// SIMATIC S7-200 project (STEP 7-Micro/WIN), CPU 226 CN REL 02.01

ORGANIZATION_BLOCK main:OB1
TITLE=自动化焊接工作站的控制程序。
// 工作站集成了传送带、预热区、焊接区和冷却区。
// 系统由启动按钮触发运行，置位运行状态标志，并通过停止按钮随时中止操作。运行状态标志只有在启动按钮被按下时才能置位，且在停止按钮按下时必须复位，确保操作员对系统状态的完全掌控。
// 焊接过程从工件传送开始。传送带电机将工件送入工作站，但只有在系统运行、工件到位传感器1和工件到位传感器2检测到工件就位，且无错误标志3、错误标志4或错误标志5时才会启动，避免工件缺失或系统故障时的误动作。
// 工件到达预热区后，预热器1开始工作，其激活条件是系统运行、特定信号满足、工件到位传感器1和工件到位传感器2确认工件到位，且无错误标志3或错误标志4，保证预热过程安全进行。预热器2在预热阶段辅助加热。预热器3在另一阶段辅助加热。预热器4在后续阶段辅助加热，以确保工件温度均匀。
// 温度控制是焊接质量的关键。系统通过温度传感器1、温度传感器2和温度传感器3实时监测预热区、焊接区和冷却区的温度，并将读数存储到温度存储变量1~3中。加热器在特定信号为1时启动。加热器应在温度低于设定值且特定信号为真时启动，以维持焊接区适宜温度。加热器在特定信号激活时开始运行。
// 焊接头和喷雾器分别在特定条件下执行操作。喷雾器需在焊接完成后启动，以冷却工件。喷雾器在特定信号触发时启动。
BEGIN
Network 1 // 网络标题
// 网络注释
LD     SM0.0
CALL   preheat1:SBR0
Network 2
LD     SM0.0
CALL   timepulse:SBR1
Network 3
LD     SM0.0
CALL   conveyor:SBR2
Network 4
LD     SM0.0
CALL   xilu:SBR3
Network 5
LD     SM0.0
CALL   preheat4:SBR4
Network 6
LD     SM0.0
CALL   pray:SBR5
Network 7
LD     SM0.0
CALL   preheat2:SBR7
Network 8
LD     SM0.0
CALL   preheat3:SBR8
Network 9
LD     SM0.0
CALL   STARTTIME:SBR9
Network 10
LD     SM0.0
CALL   state:SBR10
Network 11
LD     SM0.0
CALL   wave:SBR11
Network 12
LD     SM0.0
CALL   redlight:SBR6
Network 13
LD     SM0.0
CALL   alarm:SBR12
Network 14
LD     M20.0
EU
S      V0.0, 1
Network 15
LD     M20.1
EU
R      V0.0, 1
Network 16
LD     M20.0
TON    T120, +5
A      T120
R      M20.0, 1
Network 17
LD     M20.1
TON    T121, +5
A      T121
R      M20.1, 1
Network 18
LD     M20.2
EU
O      M0.0
AN     M20.3
AN     V828.0
AN     V828.1
AN     V880.0
=      M0.0
Network 19
LD     M20.2
TON    T122, +5
A      T122
R      M20.2, 1
Network 20
LD     M20.3
TON    T123, +5
A      T123
R      M20.3, 1
Network 21
LDN    V0.0
A      M21.7
O      V0.0
A      M0.0
A      I0.6
A      I0.7
AN     V828.4
AN     V828.2
AN     V830.1
=      Q2.5
Network 22
LD     M22.0
A      M0.0
A      I0.6
A      I0.7
AN     V828.4
AN     V828.2
=      Q1.7
Network 23
LDN    V0.0
A      M22.2
O      V0.0
A      M0.0
A      I0.6
A      I0.7
AN     V828.4
AN     V828.2
AN     V830.6
=      Q2.4
Network 24
LDN    M0.0
R      M20.5, 14
R      M22.4, 1
Network 25
LD     V0.0
R      M20.5, 5
R      M22.1, 2
R      M21.5, 1
R      M22.4, 1
Network 26
LD     V0.0
LD     M20.7
O      M21.0
O      M21.1
O      M21.2
AN     V0.0
OLD
A      M0.0
A      I0.6
A      I0.7
AN     V828.4
AN     V828.2
=      Q2.1
Network 27
LD     M22.5
=      Q0.2
Network 28
LD     M0.0
A      I0.0
EU
+I     +1, VW818
Network 29
LD     M22.3
MOVW   +0, VW818
Network 30
LD     M22.3
TON    T124, +5
A      T124
R      M22.3, 1
Network 31
LD     M22.6
MOVW   AIW10, VW812
MOVW   AIW12, VW814
MOVW   AIW14, VW816
Network 32
LD     M22.7
R      M22.6, 2
R      V822.6, 1
Network 33
LD     M22.6
=      Q1.3
S      V822.6, 1
END_ORGANIZATION_BLOCK

SUBROUTINE_BLOCK preheat1:SBR0
TITLE=子程序注释
BEGIN
Network 1 // 网络标题
// 网络注释
LD     SM0.0
MOVW   VW610, VW1500
MOVW   VW612, VW1502
MOVW   VW614, VW1504
MOVW   VW616, VW1506
Network 2
LD     SM0.0
MOVW   AIW0, VW1508
+I     VW1506, VW1508
Network 3
LDW>=  VW1508, +0
AW<=   VW1508, +2500
MOVW   VW1500, VW1510
+I     +20, VW1510
MOVW   VW1500, VW1512
+I     +5, VW1512
MOVW   VW1500, VW1514
-I     +10, VW1514
MOVW   VW1500, VW1516
-I     +15, VW1516
MOVW   VW1500, VW1518
-I     +20, VW1518
MOVW   VW1500, VW1520
-I     +25, VW1520
MOVW   VW1500, VW1522
-I     +50, VW1522
MOVW   VW1500, VW1524
-I     +100, VW1524
MOVW   VW1500, VW1542
+I     +100, VW1542
Network 4
LD     M12.0
MOVW   VW1508, VW1526
Network 5
LD     M12.2
AW>=   VW1508, VW1526
MOVW   VW1508, VW1528
-I     VW1526, VW1528
Network 6
LDW<=  VW1508, VW1524
LDW<=  VW1508, VW1526
AW<=   VW1508, VW1512
OLD
LD     M15.0
AW<=   VW1508, VW1522
AW>=   VW1508, VW1524
OLD
LD     M15.1
AW<=   VW1508, VW1520
AW>=   VW1508, VW1522
OLD
LD     M15.2
AW<=   VW1508, VW1516
AW>=   VW1508, VW1520
OLD
LDW>   VW1528, +3
A      M15.4
LDW>=  VW1528, +0
AW<=   VW1528, +3
A      M15.5
OLD
AW<=   VW1508, VW1500
AW>=   VW1508, VW1518
OLD
LD     V0.0
LDN    V0.0
A      M20.7
OLD
ALD
A      I0.6
A      I0.7
A      M0.0
AN     V825.3
AN     V828.2
AN     V828.4
AN     V880.0
=      Q1.4
Network 7
LD     V0.0
LDN    V0.0
A      M20.7
OLD
A      M0.0
OW>=   VW1508, +800
A      I0.6
A      I0.7
=      Q2.3
Network 8
LD     SM0.0
LPS
LDW<=  VW1508, VW1524
OW>    VW1508, VW1542
LDW>   VW1508, VW1514
AW<=   VW1508, VW1512
OLD
ALD
MOVW   VW1508, VW1546
LRD
AW>    VW1508, VW1524
AW<=   VW1508, VW1522
MOVW   VW1508, VW1530
AENO
+I     VW1500, VW1530
AENO
MOVW   VW1530, VW1546
/I     +2, VW1546
LPP
LDW>   VW1508, VW1522
AW<=   VW1508, VW1514
LDW>   VW1508, VW1512
AW<=   VW1508, VW1542
OLD
ALD
MOVW   VW1508, VW1532
AENO
+I     VW1500, VW1532
AENO
MOVW   VW1532, VW1534
AENO
+I     VW1500, VW1534
AENO
MOVW   VW1534, VW1546
/I     +3, VW1546
Network 9
LD     SM0.0
MOVW   VW1546, VW1548
AENO
/I     +10, VW1548
AENO
MOVW   VW1548, VW802
*I     +10, VW802
Network 10
LD     M0.0
AW<    VW802, VW1502
AW>    VW802, VW1504
=      V824.6
Network 11
LD     M0.0
AW>    VW802, VW1502
=      V825.3
END_SUBROUTINE_BLOCK

SUBROUTINE_BLOCK timepulse:SBR1
TITLE=
BEGIN
Network 1
LD     SM0.0
LPS
AN     T160
=      M15.0
LRD
AN     T161
TON    T160, +60
LPP
AN     M15.0
TON    T161, +6
Network 2
LD     SM0.0
LPS
AN     T162
=      M15.1
LRD
AN     T163
TON    T162, +35
LPP
AN     M15.1
TON    T163, +6
Network 3
LD     SM0.0
LPS
AN     T164
=      M15.2
LRD
AN     T165
TON    T164, +30
LPP
AN     M15.2
TON    T165, +6
Network 4
LD     SM0.0
LPS
AN     T166
=      M15.3
LRD
AN     T167
TON    T166, +15
LPP
AN     M15.3
TON    T167, +5
Network 5
LD     SM0.0
LPS
AN     T168
=      M15.4
LRD
AN     T169
TON    T168, +5
LPP
AN     M15.4
TON    T169, +25
Network 6
LD     SM0.0
LPS
AN     T180
=      M15.5
LRD
AN     T181
TON    T180, +10
LPP
AN     M15.5
TON    T181, +20
Network 7
LDN    M12.0
AN     M12.1
AN     M12.2
AN     M12.0
S      M12.0, 1
Network 8
LD     M12.0
TON    T182, +2
A      T182
S      M12.1, 1
R      M12.0, 1
Network 9
LD     M12.1
TON    T183, +46
A      T183
S      M12.2, 1
R      M12.1, 1
Network 10
LD     M12.2
TON    T184, +2
A      T184
R      M12.2, 1
END_SUBROUTINE_BLOCK

// SBR2: protected block, not included

// SBR3: protected block, not included

// SBR4: protected block, not included

// SBR5: protected block, not included

SUBROUTINE_BLOCK redlight:SBR6
TITLE=
BEGIN
Network 1
LD     M20.4
S      M11.0, 1
TON    T205, +5
A      T205
R      M20.4, 1
Network 2
LD     M11.0
AW=    VW828, +0
AW=    VW830, +0
R      M11.0, 1
Network 3
LDN    I0.6
S      V828.0, 1
Network 4
LD     I0.6
A      M20.4
EU
R      V828.0, 1
Network 5
LDN    I0.7
S      V828.1, 1
Network 6
LD     I0.7
A      M20.4
EU
R      V828.1, 1
Network 7
LDN    I2.3
S      V828.2, 1
Network 8
LD     I2.3
TON    T172, +50
A      T172
R      V828.2, 1
Network 9
LDN    I0.4
S      V828.4, 1
Network 10
LD     I0.4
A      M20.4
EU
R      V828.4, 1
Network 11
LDW=   VW1808, 16#7FFF
S      V828.5, 1
Network 12
LDW<   VW1808, 16#7FFF
A      M20.4
EU
R      V828.5, 1
Network 13
LDN    I2.1
S      V829.2, 1
Network 14
LD     I2.1
A      M20.4
EU
R      V829.2, 1
Network 15
LDN    I2.2
S      V829.3, 1
Network 16
LD     I2.2
A      M20.4
EU
R      V829.3, 1
Network 17
LDN    I2.4
S      V829.4, 1
Network 18
LD     I2.4
A      M20.4
EU
R      V829.4, 1
Network 19
LDN    I2.5
S      V830.1, 1
Network 20
LD     I2.5
A      M20.4
EU
R      V830.1, 1
Network 21
LDW=   VW1508, 16#7FFF
S      V830.2, 1
Network 22
LDW<   VW1508, 16#7FFF
A      M20.4
EU
R      V830.2, 1
Network 23
LDW=   VW1558, 16#7FFF
S      V830.3, 1
Network 24
LDW<   VW1558, 16#7FFF
A      M20.4
EU
R      V830.3, 1
Network 25
LDW=   VW1608, 16#7FFF
S      V830.4, 1
Network 26
LDW<   VW1608, 16#7FFF
A      M20.4
EU
R      V830.4, 1
Network 27
LDW=   VW1708, 16#7FFF
S      V830.5, 1
Network 28
LDW<   VW1708, 16#7FFF
A      M20.4
EU
R      V830.5, 1
Network 29
LDN    I1.2
S      V830.6, 1
Network 30
LD     I1.2
A      M20.4
EU
R      V830.6, 1
Network 31
LDW>   VW802, +2200
OW>    VW804, +2200
OW>    VW806, +2200
OW>    VW808, +2200
S      V831.6, 1
Network 32
LD     M20.4
EU
R      V831.6, 1
Network 33
LD     I1.5
S      V831.7, 1
Network 34
LDN    I1.5
A      M20.4
EU
R      V831.7, 1
Network 35
LDW>   VW828, +0
OW>    VW830, +0
O      V825.2
=      Q0.6
AN     M11.0
=      Q0.3
END_SUBROUTINE_BLOCK

SUBROUTINE_BLOCK preheat2:SBR7
TITLE=
BEGIN
Network 1
LD     SM0.0
MOVW   VW618, VW1550
MOVW   VW620, VW1552
MOVW   VW622, VW1554
MOVW   VW624, VW1556
Network 2
LD     SM0.0
MOVW   AIW2, VW1558
+I     VW1556, VW1558
Network 3
LDW>=  VW1558, +0
AW<=   VW1558, +2500
MOVW   VW1550, VW1560
+I     +20, VW1560
MOVW   VW1550, VW1562
+I     +5, VW1562
MOVW   VW1550, VW1564
-I     +10, VW1564
MOVW   VW1550, VW1566
-I     +15, VW1566
MOVW   VW1550, VW1568
-I     +20, VW1568
MOVW   VW1550, VW1570
-I     +25, VW1570
MOVW   VW1550, VW1572
-I     +50, VW1572
MOVW   VW1550, VW1574
-I     +100, VW1574
MOVW   VW1550, VW1592
+I     +100, VW1592
Network 4
LD     M12.0
MOVW   VW1558, VW1576
Network 5
LD     M12.2
AW>=   VW1558, VW1576
MOVW   VW1558, VW1578
-I     VW1576, VW1578
Network 6
LDW<=  VW1558, VW1574
LDW<=  VW1558, VW1576
AW<=   VW1558, VW1562
OLD
LD     M15.0
AW<=   VW1558, VW1572
AW>=   VW1558, VW1574
OLD
LD     M15.1
AW<=   VW1558, VW1570
AW>=   VW1558, VW1572
OLD
LD     M15.2
AW<=   VW1558, VW1566
AW>=   VW1558, VW1570
OLD
LDW>   VW1578, +3
A      M15.4
LDW>=  VW1578, +0
AW<=   VW1578, +3
A      M15.5
OLD
AW<=   VW1558, VW1550
AW>=   VW1558, VW1568
OLD
LD     V0.0
LDN    V0.0
A      M21.0
OLD
ALD
A      I0.6
A      I0.7
A      M0.0
AN     V825.4
AN     V828.2
AN     V828.4
AN     V880.0
=      Q1.5
Network 7
LD     V0.0
LDN    V0.0
A      M21.0
OLD
A      M0.0
OW>=   VW1558, +800
A      I0.6
A      I0.7
=      Q2.6
Network 8
LD     SM0.0
LPS
LDW<=  VW1558, VW1574
OW>    VW1558, VW1592
LDW>   VW1558, VW1564
AW<=   VW1558, VW1562
OLD
ALD
MOVW   VW1558, VW1596
LRD
AW>    VW1558, VW1574
AW<=   VW1558, VW1572
MOVW   VW1558, VW1580
AENO
+I     VW1550, VW1580
AENO
MOVW   VW1580, VW1596
/I     +2, VW1596
LPP
LDW>   VW1558, VW1572
AW<=   VW1558, VW1564
LDW>   VW1558, VW1562
AW<=   VW1558, VW1592
OLD
ALD
MOVW   VW1558, VW1582
AENO
+I     VW1550, VW1582
AENO
MOVW   VW1582, VW1584
AENO
+I     VW1550, VW1584
AENO
MOVW   VW1584, VW1596
/I     +3, VW1596
Network 9
LD     SM0.0
MOVW   VW1596, VW1598
AENO
/I     +10, VW1598
AENO
MOVW   VW1598, VW804
*I     +10, VW804
Network 10
LD     M0.0
AW<    VW804, VW1552
AW>    VW804, VW1554
=      V824.7
Network 11
LD     M0.0
AW>    VW804, VW1552
=      V825.4
Network 95
LDW<=  VW100, +320
MOVW   +180, VW120
Network 96
LDW>=  VW100, +321
AW<=   VW100, +350
MOVW   +100, VW120
END_SUBROUTINE_BLOCK

SUBROUTINE_BLOCK preheat3:SBR8
TITLE=
BEGIN
Network 1
LD     SM0.0
MOVW   VW626, VW1600
MOVW   VW628, VW1602
MOVW   VW630, VW1604
MOVW   VW632, VW1606
Network 2
LD     SM0.0
MOVW   AIW4, VW1608
+I     VW1606, VW1608
Network 3
LDW>=  VW1608, +0
AW<=   VW1608, +2500
MOVW   VW1600, VW1610
+I     +20, VW1610
MOVW   VW1600, VW1612
+I     +5, VW1612
MOVW   VW1600, VW1614
-I     +10, VW1614
MOVW   VW1600, VW1616
-I     +15, VW1616
MOVW   VW1600, VW1618
-I     +20, VW1618
MOVW   VW1600, VW1620
-I     +25, VW1620
MOVW   VW1600, VW1622
-I     +50, VW1622
MOVW   VW1600, VW1624
-I     +100, VW1624
MOVW   VW1600, VW1642
+I     +100, VW1642
Network 4
LD     M12.0
MOVW   VW1608, VW1626
Network 5
LD     M12.2
AW>=   VW1608, VW1626
MOVW   VW1608, VW1628
-I     VW1626, VW1628
Network 6
LDW<=  VW1608, VW1624
LDW<=  VW1608, VW1626
AW<=   VW1608, VW1612
OLD
LD     M15.0
AW<=   VW1608, VW1622
AW>=   VW1608, VW1624
OLD
LD     M15.1
AW<=   VW1608, VW1620
AW>=   VW1608, VW1622
OLD
LD     M15.2
AW<=   VW1608, VW1616
AW>=   VW1608, VW1620
OLD
LDW>   VW1628, +3
A      M15.4
LDW>=  VW1628, +0
AW<=   VW1628, +3
A      M15.5
OLD
AW<=   VW1608, VW1600
AW>=   VW1608, VW1618
OLD
LD     V0.0
LDN    V0.0
A      M21.1
OLD
ALD
A      I0.6
A      I0.7
A      M0.0
AN     V825.5
AN     V828.2
AN     V828.4
AN     V880.0
=      Q1.6
Network 7
LD     V0.0
LDN    V0.0
A      M21.1
OLD
A      M0.0
OW>=   VW1608, +800
A      I0.6
A      I0.7
=      Q2.7
Network 8
LD     SM0.0
LPS
LDW<=  VW1608, VW1624
OW>    VW1608, VW1642
LDW>   VW1608, VW1614
AW<=   VW1608, VW1612
OLD
ALD
MOVW   VW1608, VW1646
LRD
AW>    VW1608, VW1624
AW<=   VW1608, VW1622
MOVW   VW1608, VW1630
AENO
+I     VW1600, VW1630
AENO
MOVW   VW1630, VW1646
/I     +2, VW1646
LPP
LDW>   VW1608, VW1622
AW<=   VW1608, VW1614
LDW>   VW1608, VW1612
AW<=   VW1608, VW1642
OLD
ALD
MOVW   VW1608, VW1632
AENO
+I     VW1600, VW1632
AENO
MOVW   VW1632, VW1634
AENO
+I     VW1600, VW1634
AENO
MOVW   VW1634, VW1646
/I     +3, VW1646
Network 9
LD     SM0.0
MOVW   VW1646, VW1648
AENO
/I     +10, VW1648
AENO
MOVW   VW1648, VW806
*I     +10, VW806
Network 10
LD     M0.0
AW<    VW806, VW1602
AW>    VW806, VW1604
=      V825.0
Network 11
LD     M0.0
AW>    VW806, VW1602
=      V825.5
Network 51
LDW<=  VW100, +320
MOVW   +180, VW120
Network 52
LDW>=  VW100, +321
AW<=   VW100, +350
MOVW   +100, VW120
END_SUBROUTINE_BLOCK

// SBR9: protected block, not included

SUBROUTINE_BLOCK state:SBR10
TITLE=
BEGIN
Network 1
LD     M0.0
=      Q0.5
Network 2
LD     V0.0
=      V820.0
Network 3
LDN    V0.0
=      V820.1
Network 4
LD     M0.0
=      V820.2
Network 5
LDN    M0.0
=      V820.3
Network 6
LDN    V0.0
A      M20.5
O      V0.0
A      M0.0
OB>=   MB5, 1
=      V820.5
Network 7
LD     Q2.2
=      V820.6
Network 8
LD     Q1.4
=      V820.7
Network 9
LD     Q1.5
=      V821.0
Network 10
LD     Q1.6
=      V821.1
Network 11
LD     M21.2
=      V821.2
Network 12
LD     Q0.7
LD     V0.0
A      M21.3
OLD
=      V821.3
Network 13
LD     Q1.0
LD     V0.0
A      M21.4
OLD
=      V821.4
Network 14
LD     Q2.5
=      V821.7
Network 15
LD     Q1.7
=      V822.0
Network 16
LD     M21.6
=      V821.6
Network 17
LD     Q2.4
=      V822.2
Network 18
LD     Q0.2
=      V822.5
Network 19
LD     M21.2
=      V821.2
END_SUBROUTINE_BLOCK

// SBR11: protected block, not included

SUBROUTINE_BLOCK alarm:SBR12
TITLE=
BEGIN
Network 1
LD     Q0.0
A      Q0.2
AN     I0.2
TON    T50, +50
A      T50
S      V831.0, 1
Network 2
LD     M20.4
R      V831.0, 1
Network 3
LD     Q0.1
A      Q0.2
AN     I0.3
TON    T51, +50
A      T51
S      V831.1, 1
Network 4
LD     M20.4
R      V831.1, 1
Network 5
LD     I0.2
A      I0.3
AN     M0.0
S      V831.2, 1
Network 6
LD     M20.4
A      I0.3
AN     I0.2
R      V831.2, 1
Network 7
LD     Q2.2
A      I0.1
TON    T53, +50
A      T53
S      M17.0, 1
Network 8
LD     Q2.2
AN     I0.1
TON    T52, +30
A      T52
S      M17.1, 1
Network 9
LD     M17.0
O      M17.1
S      V831.4, 1
R      M17.0, 2
Network 10
LD     M20.4
R      V831.4, 1
R      V880.0, 1
END_SUBROUTINE_BLOCK
